Staubli VAL3: Init.pgx

public program Init()
begin
end
